FUNCTION_BLOCK FB_StateMachine
VAR_INPUT
	bStart : BOOL;
	bStop : BOOL;
	bLimitLeft : BOOL;
	bLimitRight: BOOL;
END_VAR
VAR_OUTPUT
	bMovingRight : BOOL;
	bMovingLeft: BOOL;
END_VAR
VAR
	TrigStop: R_TRIG;
	state : E_States;
	prevState : E_States;
	sState: STRING;
END_VAR

TrigStop(CLK:=bStop);

IF TrigStop.Q THEN
	prevState := state;
	state:= E_States.eStop;
END_IF	


CASE state OF
	E_States.eStop:
		sState := 'Stop';
		bMovingRight := FALSE;
		bMovingLeft := FALSE;
		IF bStart THEN
			IF prevState = E_States.eMovingLeft THEN
				state:= E_States.eMovingLeft;
			ELSE
				state:= E_States.eMovingRight;
			END_IF
		END_IF
	
	E_States.eMovingRight:
		sState := 'Moving Right';
		bMovingRight := TRUE;
		bMovingLeft := FALSE;
		IF bLimitRight THEN
			state:= E_States.eMovingLeft;
		END_IF
	
	E_States.eMovingLeft:
		sState := 'Moving Left';
		bMovingRight := FALSE;
		bMovingLeft := TRUE;
		IF bLimitLeft THEN
			state:= E_States.eMovingRight;
		END_IF
	
	
END_CASE

END_FUNCTION_BLOCK

(* stored: Version 1.1.0.1, ProductVersion 3.1.4024.12
   POU FB_StateMachine: Id {10e671e1-a6a3-45c6-a325-3335c9cdfed7}, SpecialFunc None *)
